FUNCTION_BLOCK FB_Generator_PWM
VAR_INPUT
END_VAR
VAR_OUTPUT
END_VAR
VAR
END_VAR

END_FUNCTION_BLOCK

(* stored: Version 1.1.0.1, ProductVersion 3.1.4024.13
   POU FB_Generator_PWM: Id {5ece2670-375c-49d6-b13c-78f48d48c80c}, SpecialFunc None *)
